{attribute 'qualified_only'}
VAR_GLOBAL CONSTANT
	OPEN		: BOOL := FALSE;
	CLOSED		: BOOL := TRUE;
END_VAR

(* stored: Version 1.1.0.1
   GVL VALVE_1: Id {25043e56-ee44-430c-8715-2f06ebef636c} *)
